Fanuc KAREL source: kt00761.KL

-- PROVISIONAL review KL for V770-1; original PC SHA256 b1f3b7f44547d73346c9f52792d581e8e125e34074df9a09c7537f73cad3b81e
-- Incomplete behavior may be omitted. Consult companion uncertainty JSON. Do not deploy.
PROGRAM KT00761
%NOLOCKGROUP
VAR
  I1 : INTEGER
  I2 : INTEGER
  OUT : REAL
BEGIN
  -- UNRESOLVED_PC offsets 5-16; opcodes 2E,23
  -- UNRESOLVED_PC offsets 21-32; opcodes 2E,23
  -- UNRESOLVED_PC offsets 37-48; opcodes 2E,23
  -- UNRESOLVED_PC offsets 53-64; opcodes 2E,23
  -- UNRESOLVED_PC offsets 69-86; opcodes 27,27,21,64,76,23
  -- UNRESOLVED_PC offsets 91-95; opcodes 7F
END KT00761
